FUNCTION_BLOCK FB_RectangleChild EXTENDS FB_Rectangle
VAR_INPUT
END_VAR
VAR_OUTPUT
END_VAR
VAR
END_VAR

END_FUNCTION_BLOCK

(* stored: Version 1.1.0.1, ProductVersion 3.1.4024.13
   POU FB_RectangleChild: Id {e621f85c-dffd-46a5-8c74-3e63e4e25c32}, SpecialFunc None *)
